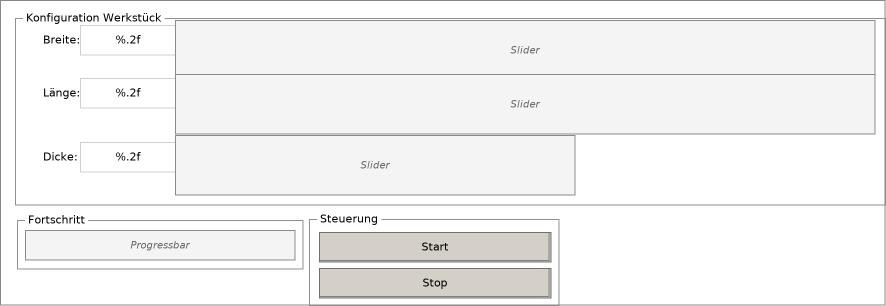
VISUALIZATION UI  // 886x306
    GroupBox (15,10 871x195), "Konfiguration Werkstück", input disabled if: GVL_Control.bIsRunning
        Label (25,15 100x30), "Breite:"
        Label (25,68 100x30), "Länge:"
        Label (25,132 100x30), "Dicke:"
        Textfield (65,15 96x30), "%.2f", text variable: GVL_Config.stConfig.rBreite
        Textfield (65,68 96x30), "%.2f", text variable: GVL_Config.stConfig.rLaenge
        Textfield (65,132 96x30), "%.2f", text variable: GVL_Config.stConfig.rDicke
        Slider (160,10 700x60), variable: GVL_Config.stConfig.rBreite, scale 300..600
        Slider (160,64 700x60), variable: GVL_Config.stConfig.rLaenge, scale 300..600
        Slider (160,125 400x60), variable: GVL_Config.stConfig.rDicke, scale 15..45
    GroupBox (17,212 286x57), "Fortschritt"
        Progressbar (8,18 270x30), variable: GVL_Control.nProgress
    GroupBox (309,211 250x95), "Steuerung"
        Button (10,21 232x30), "Start", input disabled if: GVL_Control.bIsRunning
            OnMouseClick: toggle GVL_Control.bRun
        Button (10,57 232x30), "Stop", input disabled if: (GVL_Control.bIsRunning AND NOT GVL_Control.bRun) OR NOT GVL_Control.bRun
            OnMouseClick: toggle GVL_Control.bRun
END_VISUALIZATION

(* stored: Version 1.1.0.1, ProductVersion 3.1.4024.3
   Visu UI: Id {d0d61389-f278-45a0-8d33-27aa6c8ec165} *)
